// TIA Portal V19 export
TYPE "LAF_typeInterfaceSignalsHmi"
TITLE = Interface signals HMI / Schnittstellen Signale HMI
// Structure interface signals Bool HMI / Struktur Schnittstelle Signale fuer HMI
// stored: Access Published
   STRUCT
      valueSymbolLeft : "LAF_typeInterfaceSignalsBool";   // Value symbol lleft / Werte Symbol links
      valueSymbolRight { S7_SetPoint := 'True'} : "LAF_typeInterfaceSignalsBool";   // Value symbol rght / Werte Symbol rechts
   END_STRUCT;
END_TYPE
